FUNCTION_BLOCK FB_SMPTE_TimeController IMPLEMENTS I_SMPTE_TimeController
VAR
	// Internal Time Source mode
	_eTimeSource : E_SMPTE_TimeController_Source;
	
	// Linked to TcCom Object for Time Provider if using Ext Mode
	_TcExternalTimeSource : REFERENCE TO ULINT; 
	
	// Frame Mode
	_eFrameMode: E_SMPTE_FrameMode := E_SMPTE_FrameMode.FPS_25;	// transmitting with 25 fps (frames per second)		
	
	// Used for DC Time
	_dcTime	: T_DCTIME64;
			
	// SMPTE Time Struct
	_stSMPTE_TimeStruct : ST_SMPTE_TimeStruct;
	
	// Reference time timestamp
	_bRefTimeInit : BOOL;
	
	// Current Time Strunct
	_CurrentTime :	TIMESTRUCT;
		
	// Current Time Value
	_RefTime : T_DCTIME64;
	
	// Working Time Value
	_WorkTime : T_DCTIME64;
	
	// Paused Time Value
	_PauseTime : T_DCTIME64;
	
	// Mode Status
	_eSMPTE_TimeController_Mode : E_SMPTE_TimeController_Mode;
	
	// Playing Status Variables
	_Playing : BOOL;
	
	// Paused Status Variables
	_Paused : BOOL;
	
	// Stopped Status Variables
	_Stopped : BOOL;
	
	// Reset Control Variables
	_Reset : BOOL;
	
	// Error, usually due to timesource
	_Error : BOOL;
END_VAR

METHOD AssignExternalTimeSource : BOOL
VAR_INPUT
	// Linked to TcCom Object for Time Provider if using Ext Mode
	TcExternalTimeSource : REFERENCE TO ULINT; 
END_VAR
_TcExternalTimeSource REF= TcExternalTimeSource;
AssignExternalTimeSource := TRUE;
END_METHOD

METHOD Cycle : BOOL
VAR_INST
	_CalcTimeDiff : FB_EcExtSyncCalcTimeDiff64;
	_bWasPaused : BOOL;
END_VAR
// Check Mode and compute time
CASE _eSMPTE_TimeController_Mode OF
	E_SMPTE_TimeController_Mode.Playing:
	
		// Get the working time
		UpdateTime(_WorkTime); 
		
		// Get the reference clock
		IF NOT _bRefTimeInit THEN
			_RefTime := _WorkTime;
			_bRefTimeInit := TRUE;
		END_IF
		
		// Recovery from Pause
		IF _bWasPaused THEN
			_RefTime := _WorkTime - _PauseTime;
			_bWasPaused := FALSE;
		END_IF

	E_SMPTE_TimeController_Mode.Paused:
		IF NOT _bWasPaused THEN
			_PauseTime := _WorkTime - _RefTime;
			_bWasPaused := TRUE;
		END_IF
	
	E_SMPTE_TimeController_Mode.Stopped:
		// Stop the clock and reset
		_bRefTimeInit := FALSE;
		_bWasPaused := FALSE;
		_PauseTime := 0;
		_WorkTime := 0;
		_RefTime := 0;
END_CASE

// If not paused, update the time stuct
IF NOT (_eSMPTE_TimeController_Mode = E_SMPTE_TimeController_Mode.Paused) THEN
	// Convert to time struct
	_CurrentTime := DCTIME64_TO_SYSTEMTIME(_WorkTime - _RefTime);
END_IF

// Reset
IF _Reset THEN
	_bRefTimeInit := FALSE;
	_bWasPaused := FALSE;
	_PauseTime := 0;
	_WorkTime := 0;
	_RefTime := 0;
	_Reset := FALSE;
END_IF

// Remove unused values
_CurrentTime.wDay := 0;
_CurrentTime.wDayOfWeek := 0;
_CurrentTime.wMonth := 0;
_CurrentTime.wYear := 0;
END_METHOD

PROPERTY Error : BOOL
GET
Error := _Error;
END_GET
END_PROPERTY

METHOD FB_init : BOOL
VAR_INPUT
	(* if TRUE, the retain variables are initialized (warm start / cold start)*)
	bInitRetains	: BOOL;
	(* if TRUE, the instance afterwards gets moved into the copy code (online change)*)
	bInCopyCode	: BOOL;
	(* Time Source*)
	eTimeSource	: E_SMPTE_TimeController_Source;
	(* Frame Mode, transmitting with 25 fps (frames per second) *)
	eFrameMode : E_SMPTE_FrameMode := E_SMPTE_FrameMode.FPS_25;
END_VAR
_eTimeSource := eTimeSource;
_eFrameMode := eFrameMode;
END_METHOD

(* Will pause the time*)
METHOD Pause : BOOL
VAR_INPUT
	bExecute	: BOOL;
END_VAR
VAR_INST
	rtExecute : R_TRIG;
END_VAR
rtExecute(CLK := bExecute);
IF rtExecute.Q THEN
	_eSMPTE_TimeController_Mode := E_SMPTE_TimeController_Mode.Paused;
	// Return TRUE
	Pause := TRUE;
END_IF
END_METHOD

PROPERTY Paused : BOOL
GET
Paused := _eSMPTE_TimeController_Mode = E_SMPTE_TimeController_Mode.Paused;
END_GET
END_PROPERTY

(* Starts the time*)
METHOD Play : BOOL
VAR_INPUT
	bExecute	: BOOL;
END_VAR
VAR_INST
	rtExecute :  R_TRIG;
END_VAR
rtExecute(CLK := bExecute);
IF rtExecute.Q THEN
	_eSMPTE_TimeController_Mode := E_SMPTE_TimeController_Mode.Playing;
	// Return TRUE
	Play := TRUE;
END_IF
END_METHOD

PROPERTY Playing : BOOL
GET
Playing := _eSMPTE_TimeController_Mode = E_SMPTE_TimeController_Mode.Playing;
END_GET
END_PROPERTY

(* Resets the time*)
METHOD Reset : BOOL
VAR_INPUT
	bExecute	: BOOL;
END_VAR
VAR_INST
	rtExecute :  R_TRIG;
END_VAR
rtExecute(CLK := bExecute);
IF rtExecute.Q THEN
	_Reset := TRUE;
	// Return TRUE
	Reset := TRUE;
END_IF
END_METHOD

(* Will stop the time and reset to 00:00:00:00*)
METHOD Stop : BOOL
VAR_INPUT
	bExecute	: BOOL;
END_VAR
VAR_INST
	rtExecute :  R_TRIG;
END_VAR
rtExecute(CLK := bExecute);
IF rtExecute.Q THEN
	_eSMPTE_TimeController_Mode := E_SMPTE_TimeController_Mode.Stopped;
	// Return TRUE
	Stop := TRUE;
END_IF
END_METHOD

PROPERTY Stopped : BOOL
GET
Stopped := _eSMPTE_TimeController_Mode = E_SMPTE_TimeController_Mode.Stopped;
END_GET
END_PROPERTY

(* Returns the SMPTE_TimeStruct*)
PROPERTY TimeStruct : REFERENCE TO ST_SMPTE_TimeStruct;
GET
// Compute the Time Struct for SMPTE
CASE _eFrameMode OF
	E_SMPTE_FrameMode.FPS_25:
		_stSMPTE_TimeStruct.Hours := WORD_TO_BYTE(_CurrentTime.wHour);
		_stSMPTE_TimeStruct.Minutes := WORD_TO_BYTE(_CurrentTime.wMinute);
		_stSMPTE_TimeStruct.Seconds := WORD_TO_BYTE(_CurrentTime.wSecond);
		_stSMPTE_TimeStruct.Frames := DINT_TO_BYTE(TRUNC(WORD_TO_REAL(_CurrentTime.wMilliseconds)/(1000/25)));
END_CASE

// Return the time struct
TimeStruct REF= _stSMPTE_TimeStruct;
END_GET
END_PROPERTY

METHOD INTERNAL UpdateTime: BOOL;
VAR_IN_OUT
	// Current Time Struct
	_CurDCTime : T_DCTIME64;
END_VAR
VAR_INST
	// Used for NT Time
	_ntTime	: TIMESTRUCT;
	_ntGetTime : NT_GetTime;
	// Ref Error Trig
	rtRefError : R_TRIG; 
END_VAR
// Check for reference error on External time source
rtRefError(CLK := NOT __ISVALIDREF(_TcExternalTimeSource));
IF rtRefError.Q THEN
	ADSLOGSTR( msgCtrlMask := ADSLOG_MSGTYPE_ERROR OR ADSLOG_MSGTYPE_MSGBOX, msgFmtStr := 'PLC SMPTE Time Controller: Invalid Timesource Provided or Disconnected: Use AssignExternalTimeSource()','');
END_IF

// Calculate the time
CASE _eTimeSource OF
	E_SMPTE_TimeController_Source.ExtTimeProvider:
		(* External Time Provider *)
		IF __ISVALIDREF(_TcExternalTimeSource) THEN
			_dcTime := FILETIME64_TO_DCTIME64(_TcExternalTimeSource);
			_CurDCTime := _dcTime;
			_Error := FALSE;
		ELSE
			_eSMPTE_TimeController_Mode := E_SMPTE_TimeController_Mode.Stopped;
			_Error := TRUE;
		END_IF
	
	E_SMPTE_TimeController_Source.DC_Time:
		(* External Time Provider *)
		_dcTime := F_GetCurDcTickTime64();
		_CurDCTime := _dcTime;
	
	E_SMPTE_TimeController_Source.NT_Time:
		(* NT Time Provider *)
		IF NOT _ntGetTime.BUSY THEN
			_ntGetTime(start := TRUE, TIMESTR => _ntTime);
		END_IF
		_ntGetTime(start := FALSE);
		_CurDCTime := SYSTEMTIME_TO_DCTIME64(_ntTime, 0, 0);
END_CASE

UpdateTime := TRUE;
END_METHOD

END_FUNCTION_BLOCK

(* stored: Version 1.1.0.1, ProductVersion 3.1.4024.12
   POU FB_SMPTE_TimeController: Id {f8bb69ee-4637-48a3-a2d0-76cda6a7f1f7}, SpecialFunc None
   Folder Internal: Id {2b65f861-1468-44d2-afff-c5982310faea}
   Folder Public: Id {408b811d-3e67-40c2-a780-467d316aa27d}
   Method AssignExternalTimeSource: Id {075f58a6-4c17-4017-b393-ea9de66e1cdb}
   Method Cycle: Id {390174b8-583d-4a27-8493-8f04e04b0a12}
   Property Error: Id {89e42f92-8288-46ea-85ca-9fbb5c7fda50}
   Get Get: Id {9ffa7fc2-2e0d-4231-a4b3-059f5e34fc65}
   Method FB_init: Id {5a6ff915-c3ed-4b35-953c-62882b888f89}
   Method Pause: Id {938eebb4-befc-4cdb-a04d-60e467c0199b}
   Property Paused: Id {a55c2cec-c422-4d6b-8f92-43a6f4f56a88}
   Get Get: Id {fa5d6a0b-45fa-425f-8332-a2f10fce1271}
   Method Play: Id {3fa81283-7721-4a58-8381-47eb503ec8d7}
   Property Playing: Id {e4ab9407-923c-41fa-a9fb-37f5fc227539}
   Get Get: Id {42ff8c89-15a9-4848-a3e3-809949b9725f}
   Method Reset: Id {e50c3f59-e027-470f-9b8b-a21fd6387ca6}
   Method Stop: Id {acf87e6f-9f82-4d54-8ab6-d7517a2514d9}
   Property Stopped: Id {202a74c6-2256-4db3-b2f1-9056fe5244d0}
   Get Get: Id {852fe4f2-1aa9-4432-939e-08a9a1ce66c1}
   Property TimeStruct: Id {0a0e3c00-95f7-4867-9ca7-551dddaeda42}
   Get Get: Id {d64b7452-a650-452e-b66c-a9e897a5750c}
   Method UpdateTime: Id {8c1e3179-ca55-4fb3-9925-92f1bfd8ef47} *)
